Yaskawa INFORM job: FRONT_SEARCH_0ST-2_4040_V2.JBI

/JOB
//NAME FRONT_SEARCH_0ST-2_4040_V2
///FOLDERNAME 02-SKRZYNIE_JOBS
//POS
///NPOS 175,175,0,27,0,0
///TOOL 0
///POSTYPE PULSE
///PULSE
C00000=0,-44333,40442,1,-36510,2
///LIMIT ON
C00001=0,-39199,42542,2,-34084,2
///LIMIT OFF
C00002=-31499,-58302,-23356,15027,12889,-13082
C00003=-52768,-43016,-26078,18373,38595,-18774
C00004=-77982,-19483,-4354,30116,56383,-30765
C00005=-53036,-11528,-12218,12363,64665,-17409
C00006=-53036,-11528,-12218,12363,64665,-17409
C00007=-51536,-9474,-10276,11905,64649,-16876
C00008=-51739,-9114,-7787,12104,63269,-17104
C00009=-53036,-11528,-12218,12363,64665,-17409
C00010=-17541,-26226,-24397,927,59032,-5038
C00011=-17541,-26226,-24397,927,59032,-5038
C00012=-16950,-23991,-22741,715,59568,-4818
C00013=-17036,-23563,-20101,755,58071,-4857
C00014=-17541,-26226,-24397,927,59032,-5038
C00015=34102,-23192,-21614,-15638,64271,13209
C00016=33423,-21885,-20599,-15423,64418,12942
C00017=32426,-19856,-18975,-15106,64629,12551
C00018=32578,-19611,-17013,-15290,63535,12762
C00019=33423,-21885,-20599,-15423,64418,12942
C00020=59339,-6070,-6417,-20979,72191,20891
C00021=59339,-6070,-6417,-20979,72191,20891
C00022=57897,-4256,-4562,-20702,71913,20431
C00023=58108,-3992,-2506,-20878,70835,20713
C00024=59339,-6070,-6417,-20979,72191,20891
C00025=42744,-35904,-30225,-18322,62562,16651
C00026=-53036,-11528,-12218,12363,64665,-17409
C00027=-61074,-17231,-7904,24252,52528,-22971
C00028=-61074,-17231,-7904,24252,52528,-22971
C00029=-59177,-15406,-6347,23472,52269,-22223
C00030=-59434,-14760,-3530,24018,51018,-22666
C00031=-61074,-17231,-7904,24252,52528,-22971
C00032=-21251,-33382,-19521,6074,40947,-7391
C00033=-21251,-33382,-19521,6074,40947,-7391
C00034=-20395,-31315,-18256,5488,41568,-6947
C00035=-20519,-30558,-15291,5724,40111,-7104
C00036=-21251,-33382,-19521,6074,40947,-7391
C00037=40714,-29673,-16650,-26102,50124,19151
C00038=39772,-28490,-15868,-25646,50155,18720
C00039=38397,-26644,-14604,-24971,50218,18088
C00040=38607,-26147,-12378,-25459,49238,18468
C00041=39772,-28490,-15868,-25646,50155,18720
C00042=67511,-11314,-2142,-31968,62539,26716
C00043=67511,-11314,-2142,-31968,62539,26716
C00044=65741,-9715,-638,-31574,62032,26145
C00045=66001,-9211,1712,-31967,61087,26572
C00046=67511,-11314,-2142,-31968,62539,26716
C00047=53079,-40826,-22944,-31443,50666,24588
C00048=-61074,-17231,-7904,24252,52528,-22971
C00049=-77982,-26538,-29134,27151,66629,-27745
C00050=-70983,-8594,-1966,26503,59809,-49670
C00051=-80152,19776,40785,37351,72704,-50428
C00052=-79984,20154,42529,37516,71911,-50638
C00053=-79233,18397,40079,37458,71885,-50340
C00054=-79984,20154,42529,37516,71911,-50638
C00055=-73519,23289,38838,28890,77081,-45618
C00056=-73519,24511,42682,29072,75582,-46027
C00057=-73519,23289,38838,28890,77081,-45618
C00058=-88897,15706,42282,50101,71325,-56974
C00059=-88897,15706,42282,50101,71325,-56974
C00060=-87612,12343,37838,50071,70996,-56519
C00061=-85283,14202,40272,50301,69633,-56165
C00062=-87338,12550,38107,50098,70839,-56476
C00063=-87612,12343,37838,50071,70996,-56519
C00064=-85283,14202,40272,50301,69633,-56165
C00065=-85878,13706,39619,50242,69986,-56252
C00066=-87297,17368,44552,50306,70316,-56776
C00067=-86572,18002,45430,50395,69865,-56680
C00068=-86135,16824,43807,50366,69783,-56505
C00069=-86572,18002,45430,50395,69865,-56680
C00070=-88872,24341,63776,52472,66292,-60220
C00071=-88146,25107,64959,52661,65790,-60187
C00072=-86432,27081,68061,53148,64560,-60149
C00073=-71828,24818,39377,28050,77174,-44632
C00074=-71828,26631,45090,28323,74925,-45226
C00075=-71828,24818,39377,28050,77174,-44632
C00076=-76970,18053,29854,27974,80136,-45734
C00077=-84952,-1789,13569,34660,47724,-58955
C00078=-67641,-1674,11109,10330,44856,-44725
C00079=-66443,961,13975,9688,44721,-44210
C00080=-67641,-1674,11109,10330,44856,-44725
C00081=-67641,-376,15347,10694,42950,-44967
C00082=-67641,-1674,11109,10330,44856,-44725
C00083=-79040,417,20398,15965,28992,-57786
C00084=-76655,5212,30978,15501,25024,-57306
C00085=-76655,6949,35816,16758,23084,-57955
C00086=-76655,5212,30978,15501,25024,-57306
C00087=-74761,6919,33010,13466,24593,-56049
C00088=-80460,-2874,12270,15804,32253,-57809
C00089=-61258,-29124,-13156,26560,43617,-22150
C00090=-51617,-32683,-18184,26745,46624,-10477
C00091=-46065,-21275,-16818,14410,65170,-6472
C00092=-47312,-18677,-12431,14817,64360,-7027
C00093=-47312,-18091,-10360,14937,63410,-7161
C00094=-47312,-18145,-10549,14927,63496,-7148
C00095=-45835,-16139,-8853,14546,63567,-6606
C00096=-47312,-18515,-11853,14850,64094,-7064
C00097=-28049,-29813,-20248,10248,58487,-729
C00098=-27208,-29156,-17681,10147,57131,-553
C00099=-27208,-28314,-15094,10280,56002,-667
C00100=-27208,-28414,-15400,10264,56134,-654
C00101=-25920,-25747,-13558,9807,56708,-112
C00102=-28049,-29813,-20248,10248,58487,-729
C00103=-30420,-40507,-29240,27153,53235,15188
C00104=-18589,-38725,-21450,23338,47896,18931
C00105=-17722,-35233,-16455,23322,46926,19051
C00106=-17722,-33749,-12435,23948,45421,18620
C00107=-17722,-33892,-12819,23887,45564,18661
C00108=-16677,-31133,-11209,23138,46167,19311
C00109=-17819,-35820,-17540,23246,47228,19090
C00110=-74104,-11494,-6266,31916,75042,4269
C00111=-71226,-7329,2631,32115,71468,4273
C00112=-71226,-6504,5446,32343,70365,3922
C00113=-71226,-6611,5086,32313,70505,3967
C00114=-68386,-4058,7675,32040,69573,4789
C00115=-73314,-9412,-353,32206,72648,3829
C00116=12839,-39975,-26573,8862,44285,32145
C00117=13766,-35291,-15908,9020,40413,32143
C00118=13766,-33973,-12356,9296,38979,31975
C00119=13766,-34084,-12651,9272,39098,31990
C00120=12880,-31062,-10895,9553,40249,31711
C00121=13449,-34253,-15344,9121,40837,32046
C00122=34752,-32856,-20023,-2690,44314,41776
C00123=37826,-27693,-13000,-4375,43497,43167
C00124=37826,-26989,-10911,-4449,42591,43216
C00125=37826,-27078,-11174,-4439,42705,43210
C00126=36403,-25075,-9779,-3633,43182,42550
C00127=37387,-27313,-13262,-4106,43940,42952
C00128=51751,-31069,-22965,-10739,49070,48663
C00129=49028,-23852,-11575,-9841,46366,47823
C00130=49028,-23004,-8935,-10039,45204,47956
C00131=49028,-23118,-9286,-10013,45357,47939
C00132=47000,-20813,-7527,-8928,45644,47024
C00133=50476,-26208,-15307,-10408,47325,48332
C00134=90602,-5375,6902,-38786,69848,59444
C00135=83174,19950,50269,-44999,67580,58220
C00136=82362,17902,47383,-44926,67511,57879
C00137=83515,19072,48341,-44798,68200,58056
C00138=78091,19382,40247,-36371,72286,52960
C00139=78091,20664,44011,-36670,70997,53443
C00140=78091,19382,40247,-36371,72286,52960
C00141=88699,7296,38566,-55615,63182,60372
C00142=86803,3068,32674,-55410,62638,59657
C00143=84852,4315,34115,-55564,61561,59330
C00144=86803,3068,32674,-55410,62638,59657
C00145=86802,3071,32670,-55412,62637,59656
C00146=84841,4323,34118,-55565,61556,59328
C00147=85129,4132,33896,-55543,61716,59376
C00148=86865,7584,38019,-55524,62521,59791
C00149=86411,7896,38400,-55569,62261,59723
C00150=85729,6493,36690,-55567,61959,59548
C00151=90097,7310,37680,-55261,64265,60355
C00152=90097,12399,50961,-57428,61452,62682
C00153=88955,13199,52025,-57644,60784,62554
C00154=86753,14877,54296,-58085,59469,62330
C00155=88537,13503,52431,-57727,60536,62506
C00156=68238,9730,17142,-24521,72673,41729
C00157=68238,11669,24062,-24961,69688,42422
C00158=72523,-3583,3802,-23332,61409,48169
C00159=73393,-10627,10934,-27897,30744,62458
C00160=70789,-6606,18800,-27824,27830,62140
C00161=69654,-4593,20814,-26755,27596,61444
C00162=70789,-6606,18800,-27824,27830,62140
C00163=70789,-5070,23059,-29482,26284,63017
C00164=70789,-6606,18800,-27824,27830,62140
C00165=83486,-8736,6503,-27040,35338,66550
C00166=77831,-2041,26192,-25270,18452,68895
C00167=77967,1961,32070,-26860,17569,69698
C00168=77967,5243,40752,-32914,14549,72656
C00169=77967,1961,32070,-26860,17569,69698
C00170=74560,4730,35257,-21622,16551,66717
C00171=77967,1961,32070,-26860,17569,69698
C00172=81109,-22356,2664,-22493,33121,60116
C00173=86168,-49730,-13668,-23926,46819,49343
C00174=44183,-52048,-7537,-24795,46064,51426
BC00000=703576
BC00001=725656
BC00002=743487
BC00003=743487
BC00004=743487
BC00005=758848
BC00006=758848
BC00007=758848
BC00008=758848
BC00009=758848
BC00010=758848
BC00011=758848
BC00012=758848
BC00013=758848
BC00014=758848
BC00015=758848
BC00016=758848
BC00017=758848
BC00018=758848
BC00019=758848
BC00020=758848
BC00021=758848
BC00022=758848
BC00023=758848
BC00024=758848
BC00025=758848
BC00026=758848
BC00027=752704
BC00028=752704
BC00029=752704
BC00030=752704
BC00031=752704
BC00032=752704
BC00033=752704
BC00034=752704
BC00035=752704
BC00036=752704
BC00037=752704
BC00038=752704
BC00039=752704
BC00040=752704
BC00041=752704
BC00042=752704
BC00043=752704
BC00044=752704
BC00045=752704
BC00046=752704
BC00047=752704
BC00048=752704
BC00049=758848
BC00050=758848
BC00051=758848
BC00052=758850
BC00053=758850
BC00054=758850
BC00055=758850
BC00056=758850
BC00057=758850
BC00058=758850
BC00059=758850
BC00060=758850
BC00061=758850
BC00062=758850
BC00063=758850
BC00064=758850
BC00065=758850
BC00066=758850
BC00067=758850
BC00068=758850
BC00069=758850
BC00070=758847
BC00071=758847
BC00072=758847
BC00073=758847
BC00074=758847
BC00075=758847
BC00076=758847
BC00077=758850
BC00078=758850
BC00079=758850
BC00080=758850
BC00081=758850
BC00082=758850
BC00083=758850
BC00084=758850
BC00085=758850
BC00086=758850
BC00087=758850
BC00088=758850
BC00089=758851
BC00090=758851
BC00091=758851
BC00092=758851
BC00093=758851
BC00094=758851
BC00095=758851
BC00096=758851
BC00097=758850
BC00098=758850
BC00099=758850
BC00100=758850
BC00101=758850
BC00102=758850
BC00103=758852
BC00104=758852
BC00105=758852
BC00106=758852
BC00107=758852
BC00108=758852
BC00109=758852
BC00110=758852
BC00111=758852
BC00112=758852
BC00113=758852
BC00114=758824
BC00115=758838
BC00116=758838
BC00117=758838
BC00118=758838
BC00119=758838
BC00120=758838
BC00121=758838
BC00122=758838
BC00123=758838
BC00124=758838
BC00125=758838
BC00126=758838
BC00127=758838
BC00128=758838
BC00129=758838
BC00130=758838
BC00131=758838
BC00132=758838
BC00133=758838
BC00134=758852
BC00135=758852
BC00136=758852
BC00137=758852
BC00138=758852
BC00139=758852
BC00140=758852
BC00141=758852
BC00142=758852
BC00143=758852
BC00144=758852
BC00145=758849
BC00146=758849
BC00147=758849
BC00148=758849
BC00149=758849
BC00150=758849
BC00151=758849
BC00152=758849
BC00153=758849
BC00154=758849
BC00155=758849
BC00156=758849
BC00157=758849
BC00158=758850
BC00159=758852
BC00160=758852
BC00161=758852
BC00162=758852
BC00163=758852
BC00164=758852
BC00165=758852
BC00166=758852
BC00167=758852
BC00168=758852
BC00169=758852
BC00170=758852
BC00171=758852
BC00172=727067
BC00173=700622
BC00174=653841
///POSTYPE BASE
///RECTAN
///RCONF 1,0,0,0,0,0,0,0,0,0,0,0,0,0,0,0,0,0,0,0,0,0,0,0
P00006=0.000,0.000,0.000,0.0000,0.0000,0.0000
///RCONF 0,0,0,0,0,0,0,0,0,0,0,0,0,0,0,0,0,0,0,0,0,0,0,0
P00021=6.550,-0.003,-5.735,0.0000,0.0000,0.0000
P00022=5.943,-0.018,-6.388,0.0000,0.0000,0.0000
P00023=7.025,-0.019,-7.168,0.0000,0.0000,0.0000
P00024=5.926,-0.047,-4.777,0.0000,0.0000,0.0000
P00058=0.000,0.000,3.000,0.0000,0.0000,0.0000
P00350=11.519,-0.008,1.149,0.0000,0.0000,0.0000
P00351=13.563,-0.027,-0.653,0.0000,0.0000,0.0000
P00352=13.252,-0.027,-0.827,0.0000,0.0000,0.0000
P00353=10.971,-0.082,0.776,0.0000,0.0000,0.0000
P00399=-2.449,0.031,8.825,0.0000,0.0000,0.0000
P00400=5.920,-3.503,-0.024,0.0000,0.0000,0.0000
P00401=3.430,-0.021,1.131,0.0000,0.0000,0.0000
P00402=-0.253,1.107,3.062,0.0000,0.0000,0.0000
P00403=-3.666,-0.015,5.328,0.0000,0.0000,0.0000
P00405=2.420,0.007,1.427,0.0000,0.0000,0.0000
P00406=3.513,-0.022,0.429,0.0000,0.0000,0.0000
P00415=-1.781,-1.303,3.250,0.0000,0.0000,0.0000
P00416=0.027,1.119,3.078,0.0000,0.0000,0.0000
P00420=-0.017,0.555,2.209,0.0000,0.0000,0.0000
P00421=4.378,0.044,2.315,0.0000,0.0000,0.0000
P00422=2.474,0.026,-1.450,0.0000,0.0000,0.0000
P00423=4.044,0.004,-2.619,0.0000,0.0000,0.0000
P00424=-0.387,-0.003,1.304,0.0000,0.0000,0.0000
P00425=-1.050,0.029,1.708,0.0000,0.0000,0.0000
P00426=0.002,-0.749,-0.024,0.0000,0.0000,0.0000
P00427=-1.030,-0.025,3.232,0.0000,0.0000,0.0000
//INST
///DATE 2025/03/10 11:44
///ATTR SC,RW
///GROUP1 RB1,BS1
NOP
MOVJ C00000 BC00000 VJ=30.00
MOVJ C00001 BC00001 VJ=20.00
MOVJ C00002 BC00002 VJ=20.00
MOVJ C00003 BC00003 VJ=20.00
MOVJ C00004 BC00004 VJ=10.00
'DODANE
'SZUKANIE FRONT
'------------------------
'503
'------------------------
MOVL C00005 BC00005 V=166.7
MOVL C00006 BC00006 V=66.7 PL=0
REFP 3 C00007 BC00007
CALL JOB:SEARCH-R1
IMOV P0058 V=16.7
SET P0350 P0006
SFTON P0350
REFP 3 C00008 BC00008
CALL JOB:SEARCH-R1
SET P0350 P0006
SFTON P0350
MOVL C00009 BC00009 V=66.7 PL=0
SFTOF
'------------------------
'------------------------
'502
'------------------------
MOVL C00010 BC00010 V=166.7
MOVL C00011 BC00011 V=66.7 PL=0
REFP 3 C00012 BC00012
CALL JOB:SEARCH-R1
IMOV P0058 V=16.7
SET P0351 P0006
SFTON P0351
REFP 3 C00013 BC00013
CALL JOB:SEARCH-R1
SET P0351 P0006
SFTON P0351
MOVL C00014 BC00014 V=66.7 PL=0
SFTOF
'------------------------
'------------------------
'501
'------------------------
MOVL C00015 BC00015 V=166.7
MOVL C00016 BC00016 V=66.7 PL=0
REFP 3 C00017 BC00017
CALL JOB:SEARCH-R1
IMOV P0058 V=16.7
SET P0352 P0006
SFTON P0352
REFP 3 C00018 BC00018
CALL JOB:SEARCH-R1
SET P0352 P0006
SFTON P0352
MOVL C00019 BC00019 V=66.7 PL=0
SFTOF
'------------------------
'------------------------
'500
'------------------------
MOVL C00020 BC00020 V=166.7
MOVL C00021 BC00021 V=66.7 PL=0
REFP 3 C00022 BC00022
CALL JOB:SEARCH-R1
IMOV P0058 V=16.7
SET P0353 P0006
SFTON P0353
REFP 3 C00023 BC00023
CALL JOB:SEARCH-R1
SET P0353 P0006
SFTON P0353
MOVL C00024 BC00024 V=66.7 PL=0
SFTOF
'------------------------
MOVL C00025 BC00025 V=333.3
MOVL C00026 BC00026 V=333.3
'NOWY
MOVL C00027 BC00027 V=166.7
MOVL C00028 BC00028 V=166.7 PL=0
REFP 3 C00029 BC00029
CALL JOB:SEARCH-R1
IMOV P0058 V=16.7
SET P0021 P0006
SFTON P0021
REFP 3 C00030 BC00030
CALL JOB:SEARCH-R1
SET P0021 P0006
SFTON P0021
MOVL C00031 BC00031 V=166.7 PL=0
SFTOF
'------------------------
'------------------------
'502
'------------------------
MOVL C00032 BC00032 V=166.7
MOVL C00033 BC00033 V=166.7 PL=0
REFP 3 C00034 BC00034
CALL JOB:SEARCH-R1
IMOV P0058 V=16.7
SET P0022 P0006
SFTON P0022
REFP 3 C00035 BC00035
CALL JOB:SEARCH-R1
SET P0022 P0006
SFTON P0022
MOVL C00036 BC00036 V=166.7 PL=0
SFTOF
'------------------------
'------------------------
'501
'------------------------
MOVL C00037 BC00037 V=166.7
MOVL C00038 BC00038 V=166.7 PL=0
REFP 3 C00039 BC00039
CALL JOB:SEARCH-R1
IMOV P0058 V=16.7
SET P0023 P0006
SFTON P0023
REFP 3 C00040 BC00040
CALL JOB:SEARCH-R1
SET P0023 P0006
SFTON P0023
MOVL C00041 BC00041 V=166.7 PL=0
SFTOF
'------------------------
'------------------------
'500
'------------------------
MOVL C00042 BC00042 V=166.7
MOVL C00043 BC00043 V=166.7 PL=0
REFP 3 C00044 BC00044
CALL JOB:SEARCH-R1
IMOV P0058 V=16.7
SET P0024 P0006
SFTON P0024
REFP 3 C00045 BC00045
CALL JOB:SEARCH-R1
SET P0024 P0006
SFTON P0024
MOVL C00046 BC00046 V=166.7 PL=0
SFTOF
'------------------------
MOVL C00047 BC00047 V=333.3
MOVL C00048 BC00048 V=333.3
MOVJ C00049 BC00049 VJ=10.00
'DODANE
MOVJ C00050 BC00050 VJ=10.00
'------------------------
'SFT402
'------------------------
SFTOF
MOVL C00051 BC00051 V=150.0
MOVL C00052 BC00052 V=166.7 PL=0
REFP 3 C00053 BC00053
CALL JOB:SEARCH-R1
SET P0402 P0006
SFTON P0402
MOVL C00054 BC00054 V=150.0
MOVL C00055 BC00055 V=66.7 PL=0
REFP 3 C00056 BC00056
CALL JOB:SEARCH-R1
SET P0402 P0006
SFTON P0402
MOVL C00057 BC00057 V=133.3
MOVL C00058 BC00058 V=150.0
MOVL C00059 BC00059 V=150.0
MOVL C00060 BC00060 V=66.7 PL=0
REFP 3 C00061 BC00061
CALL JOB:SEARCH-R1
SET P0402 P0006
SFTOF
MOVL C00062 BC00062 V=150.0
'------------------------
'SFT403
'------------------------
'START
SFTOF
MOVL C00063 BC00063 V=66.7 PL=0
REFP 3 C00064 BC00064
CALL JOB:SEARCH-R1
SET P0420 P0006
SFTON P0420
MOVL C00065 BC00065 V=150.0
MOVL C00066 BC00066 V=250.0
MOVL C00067 BC00067 V=133.3 PL=0
REFP 3 C00068 BC00068
CALL JOB:SEARCH-R1
SET P0420 P0006
SFTON P0420
MOVL C00069 BC00069 V=133.3
SFTOF
MOVL C00070 BC00070 V=250.0
MOVL C00071 BC00071 V=133.3 PL=0
REFP 3 C00072 BC00072
CALL JOB:SEARCH-R1
SET P0421 P0006
SFTON P0421
MOVL C00073 BC00073 V=133.3
REFP 3 C00074 BC00074
CALL JOB:SEARCH-R1
SET P0421 P0006
SFTON P0421
MOVL C00075 BC00075 V=133.3
MOVL C00076 BC00076 V=250.0
SFTOF
MOVL C00077 BC00077 V=250.0
MOVL C00078 BC00078 V=133.3 PL=0
REFP 3 C00079 BC00079
CALL JOB:SEARCH-R1
SET P0416 P0006
SFTON P0416
MOVL C00080 BC00080 V=133.3
REFP 3 C00081 BC00081
CALL JOB:SEARCH-R1
SET P0402 P0006
SFTOF
MOVL C00082 BC00082 V=150.0
'------------------------
'------------------------
SFTOF
MOVL C00083 BC00083 V=250.0
MOVL C00084 BC00084 V=133.3 PL=0
REFP 3 C00085 BC00085
CALL JOB:SEARCH-R1
SET P0403 P0006
SFTON P0403
MOVL C00086 BC00086 V=66.7 PL=0
REFP 3 C00087 BC00087
CALL JOB:SEARCH-R1
SET P0403 P0006
SFTOF
MOVL C00088 BC00088 V=150.0
MOVJ C00089 BC00089 VJ=20.00
MOVJ C00090 BC00090 VJ=20.00
MOVL C00091 BC00091 V=250.0
MOVL C00092 BC00092 V=133.3 PL=0
REFP 3 C00093 BC00093
CALL JOB:SEARCH-R1
SET P0422 P0006
SFTON P0422
MOVL C00094 BC00094 V=66.7 PL=0
REFP 3 C00095 BC00095
CALL JOB:SEARCH-R1
SET P0422 P0006
SFTOF
MOVL C00096 BC00096 V=250.0
MOVL C00097 BC00097 V=250.0
MOVL C00098 BC00098 V=133.3 PL=0
REFP 3 C00099 BC00099
CALL JOB:SEARCH-R1
SET P0423 P0006
SFTON P0423
MOVL C00100 BC00100 V=66.7 PL=0
REFP 3 C00101 BC00101
CALL JOB:SEARCH-R1
SET P0423 P0006
SFTOF
MOVL C00102 BC00102 V=250.0
MOVJ C00103 BC00103 VJ=20.00
'------------------------
'SFT401
'------------------------
SFTOF
MOVL C00104 BC00104 V=150.0
MOVL C00105 BC00105 V=66.7 PL=0
REFP 3 C00106 BC00106
CALL JOB:SEARCH-R1
SET P0401 P0006
SFTON P0401
MOVL C00107 BC00107 V=66.7 PL=0
REFP 3 C00108 BC00108
CALL JOB:SEARCH-R1
SET P0401 P0006
SFTOF
MOVL C00109 BC00109 V=150.0
'SFT400
'------------------------
SFTOF
MOVL C00110 BC00110 V=333.3
MOVL C00111 BC00111 V=66.7 PL=0
REFP 3 C00112 BC00112
CALL JOB:SEARCH-R1
SET P0405 P0006
SFTON P0405
MOVL C00113 BC00113 V=66.7 PL=0
REFP 3 C00114 BC00114
CALL JOB:SEARCH-R1
SET P0405 P0006
SFTOF
MOVL C00115 BC00115 V=150.0
'SFT400
'------------------------
SFTOF
MOVL C00116 BC00116 V=250.0
MOVL C00117 BC00117 V=133.3 PL=0
REFP 3 C00118 BC00118
CALL JOB:SEARCH-R1
SET P0424 P0006
SFTON P0424
MOVL C00119 BC00119 V=66.7 PL=0
REFP 3 C00120 BC00120
CALL JOB:SEARCH-R1
SET P0424 P0006
SFTOF
MOVL C00121 BC00121 V=250.0
MOVL C00122 BC00122 V=250.0
MOVL C00123 BC00123 V=133.3 PL=0
REFP 3 C00124 BC00124
CALL JOB:SEARCH-R1
SET P0425 P0006
SFTON P0425
MOVL C00125 BC00125 V=66.7 PL=0
REFP 3 C00126 BC00126
CALL JOB:SEARCH-R1
SET P0425 P0006
SFTOF
MOVL C00127 BC00127 V=250.0
MOVL C00128 BC00128 V=333.3
MOVL C00129 BC00129 V=133.3 PL=0
REFP 3 C00130 BC00130
CALL JOB:SEARCH-R1
SET P0406 P0006
SFTON P0406
MOVL C00131 BC00131 V=66.7 PL=0
REFP 3 C00132 BC00132
CALL JOB:SEARCH-R1
SET P0406 P0006
SFTOF
MOVL C00133 BC00133 V=150.0
'SFT400
'------------------------
SFTOF
MOVL C00134 BC00134 V=150.0
MOVL C00135 BC00135 V=66.7 PL=0
REFP 3 C00136 BC00136
CALL JOB:SEARCH-R1
SET P0400 P0006
SFTON P0400
MOVL C00137 BC00137 V=150.0
MOVL C00138 BC00138 V=66.7 PL=0
REFP 3 C00139 BC00139
CALL JOB:SEARCH-R1
SET P0400 P0006
SFTON P0400
MOVL C00140 BC00140 V=150.0
MOVL C00141 BC00141 V=150.0
MOVL C00142 BC00142 V=66.7 PL=0
REFP 3 C00143 BC00143
CALL JOB:SEARCH-R1
SET P0400 P0006
SFTOF
MOVL C00144 BC00144 V=83.3
MOVL C00145 BC00145 V=133.3 PL=0
REFP 3 C00146 BC00146
CALL JOB:SEARCH-R1
SET P0426 P0006
SFTON P0426
MOVL C00147 BC00147 V=66.7 PL=0
MOVL C00148 BC00148 V=166.7
MOVL C00149 BC00149 V=166.7
REFP 3 C00150 BC00150
CALL JOB:SEARCH-R1
SET P0426 P0006
SFTOF
MOVL C00151 BC00151 V=250.0
MOVL C00152 BC00152 V=250.0
MOVL C00153 BC00153 V=133.3 PL=0
REFP 3 C00154 BC00154
CALL JOB:SEARCH-R1
SET P0427 P0006
SFTON P0427
MOVL C00155 BC00155 V=66.7 PL=0
MOVL C00156 BC00156 V=166.7
REFP 3 C00157 BC00157
CALL JOB:SEARCH-R1
SET P0427 P0006
SFTOF
MOVL C00158 BC00158 V=250.0
MOVL C00159 BC00159 V=333.3
MOVL C00160 BC00160 V=66.7 PL=0
REFP 3 C00161 BC00161
CALL JOB:SEARCH-R1
SET P0415 P0006
SFTON P0415
MOVL C00162 BC00162 V=133.3
REFP 3 C00163 BC00163
CALL JOB:SEARCH-R1
SET P0415 P0006
SFTOF
MOVL C00164 BC00164 V=150.0
'------------------------
'SFT403
'------------------------
'START
SFTOF
MOVJ C00165 BC00165 VJ=10.00
'------------------------
'SFT399
'------------------------
'START
SFTOF
MOVL C00166 BC00166 V=150.0
MOVL C00167 BC00167 V=66.7 PL=0
REFP 3 C00168 BC00168
CALL JOB:SEARCH-R1
SET P0399 P0006
SFTON P0399
MOVL C00169 BC00169 V=66.7 PL=0
REFP 3 C00170 BC00170
CALL JOB:SEARCH-R1
SET P0399 P0006
SFTOF
MOVL C00171 BC00171 V=150.0
MOVJ C00172 BC00172 VJ=20.00
MOVJ C00173 BC00173 VJ=30.00
MOVJ C00174 BC00174 VJ=30.00
END
